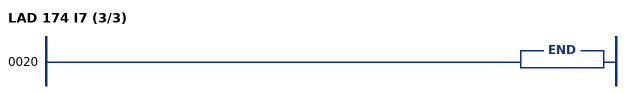
% Rung: 20 %
SOR END EOR

LADDER 175 "I7 RESULT"
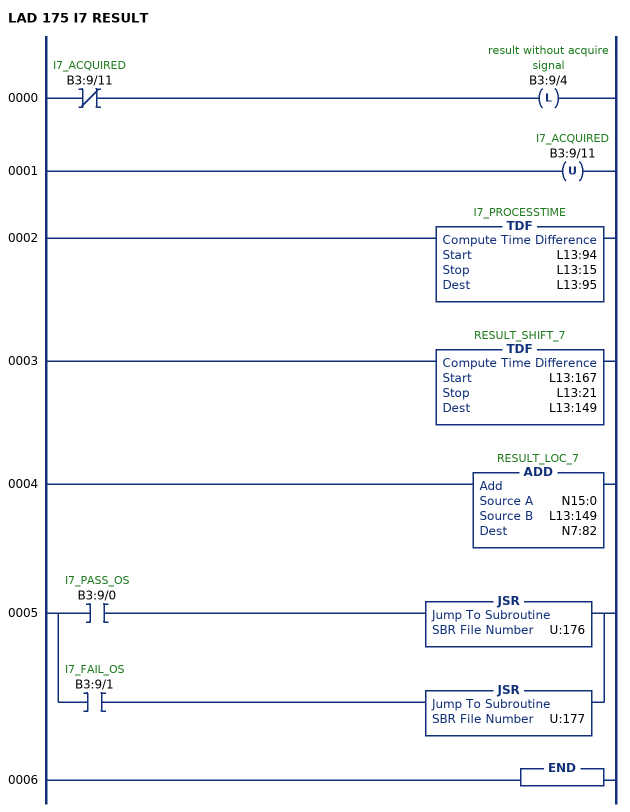
% Rung: 0 %
SOR XIO B3:9/11 OTL B3:9/4 EOR
%   B3:9/11  I7_ACQUIRED %
%   B3:9/4  "result without acquire signal" %
% Rung: 1 %
SOR OTU B3:9/11 EOR
%   B3:9/11  I7_ACQUIRED %
% Rung: 2 %
SOR TDF L13:94 L13:15 L13:95 EOR
%   L13:94  I7_TIMEOFACQ %
%   L13:15  THE_TIME %
%   L13:95  I7_PROCESSTIME %
% Rung: 3 %
SOR TDF L13:167 L13:21 L13:149 EOR
%   L13:167  I7_PROCESS_START_POS %
%   L13:21  TOP_POSITION %
%   L13:149  RESULT_SHIFT_7 %
% Rung: 4 %
SOR ADD N15:0 L13:149 N7:82 EOR
%   N15:0  I7_TRIG_LOC %
%   L13:149  RESULT_SHIFT_7 %
%   N7:82  RESULT_LOC_7 %
% Rung: 5 %
SOR BST XIC B3:9/0 JSR U:176 NXB XIC B3:9/1 JSR U:177 BND EOR
%   B3:9/0  I7_PASS_OS %
%   B3:9/1  I7_FAIL_OS %
% Rung: 6 %
SOR END EOR

LADDER 176 "I7 PASS"
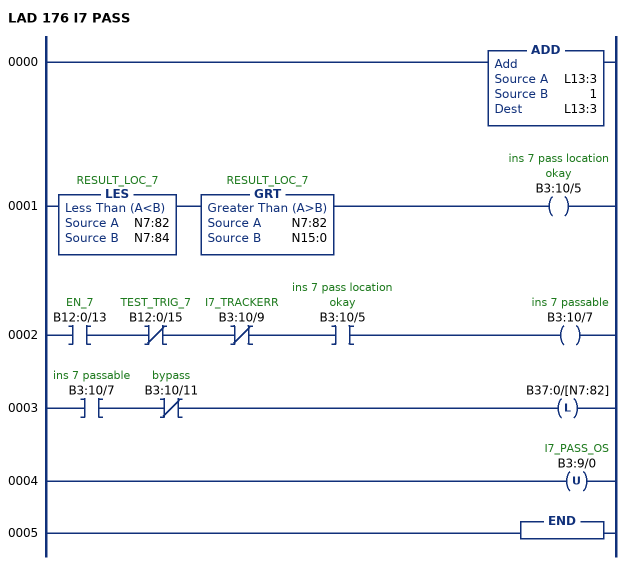
% Rung: 0 %
SOR ADD L13:3 1 L13:3 EOR
% Rung: 1 %
SOR LES N7:82 N7:84 GRT N7:82 N15:0 OTE B3:10/5 EOR
%   N7:82  RESULT_LOC_7 %
%   N7:84  I7_MAX_SHIFT %
%   N15:0  I7_TRIG_LOC %
%   B3:10/5  "ins 7 pass location okay" %
% Rung: 2 %
SOR XIC B12:0/13 XIO B12:0/15 XIO B3:10/9 XIC B3:10/5 OTE B3:10/7 EOR
%   B12:0/13  EN_7 %
%   B12:0/15  TEST_TRIG_7 %
%   B3:10/9  I7_TRACKERR %
%   B3:10/5  "ins 7 pass location okay" %
%   B3:10/7  "ins 7 passable" %
% Rung: 3 %
SOR XIC B3:10/7 XIO B3:10/11 OTL B37:0/[N7:82] EOR
%   B3:10/7  "ins 7 passable" %
%   B3:10/11  "bypass" %
%   B37:0  TOPGOOD1 %
%   N7:82  RESULT_LOC_7 %
% Rung: 4 %
SOR OTU B3:9/0 EOR
%   B3:9/0  I7_PASS_OS %
% Rung: 5 %
SOR END EOR

LADDER 177 "I7 FAIL"
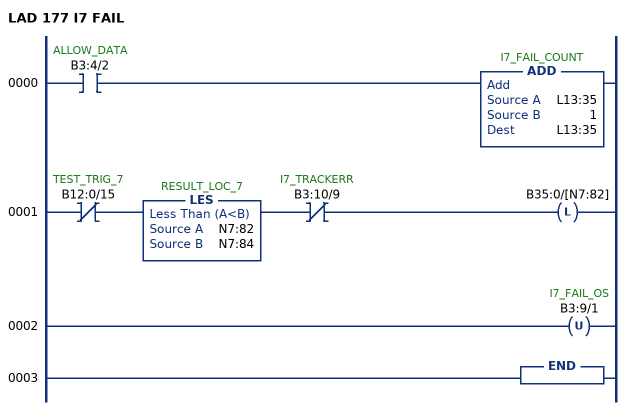
% Rung: 0 %
SOR XIC B3:4/2 ADD L13:35 1 L13:35 EOR
%   B3:4/2  ALLOW_DATA %
%   L13:35  I7_FAIL_COUNT %
% Rung: 1 %
SOR XIO B12:0/15 LES N7:82 N7:84 XIO B3:10/9 OTL B35:0/[N7:82] EOR
%   B12:0/15  TEST_TRIG_7 %
%   N7:82  RESULT_LOC_7 %
%   N7:84  I7_MAX_SHIFT %
%   B3:10/9  I7_TRACKERR %
%   B35:0  TOP_NG %
% Rung: 2 %
SOR OTU B3:9/1 EOR
%   B3:9/1  I7_FAIL_OS %
% Rung: 3 %
SOR END EOR

LADDER 178 "I7 ACQ"
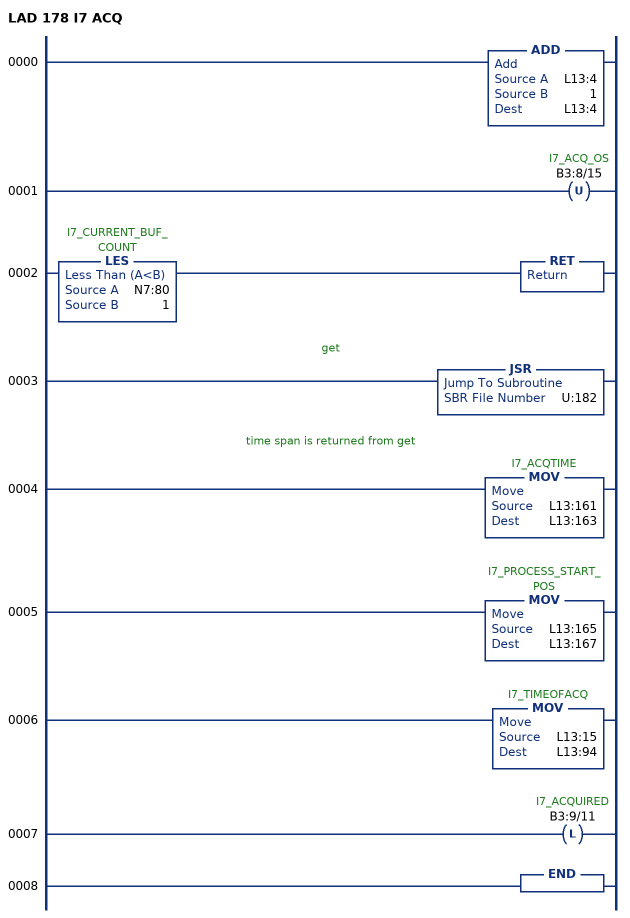
% Rung: 0 %
SOR ADD L13:4 1 L13:4 EOR
% Rung: 1 %
SOR OTU B3:8/15 EOR
%   B3:8/15  I7_ACQ_OS %
% Rung: 2 %
SOR LES N7:80 1 RET EOR
%   N7:80  I7_CURRENT_BUF_COUNT %
% Rung: 3 %
% get %
SOR JSR U:182 EOR
% Rung: 4 %
% time span is returned from get %
SOR MOV L13:161 L13:163 EOR
%   L13:161  I7_TIME_SPAN %
%   L13:163  I7_ACQTIME %
% Rung: 5 %
SOR MOV L13:165 L13:167 EOR
%   L13:165  I7_PULLED_POSITION %
%   L13:167  I7_PROCESS_START_POS %
% Rung: 6 %
SOR MOV L13:15 L13:94 EOR
%   L13:15  THE_TIME %
%   L13:94  I7_TIMEOFACQ %
% Rung: 7 %
SOR OTL B3:9/11 EOR
%   B3:9/11  I7_ACQUIRED %
% Rung: 8 %
SOR END EOR

LADDER 179 "I7 TESTER"
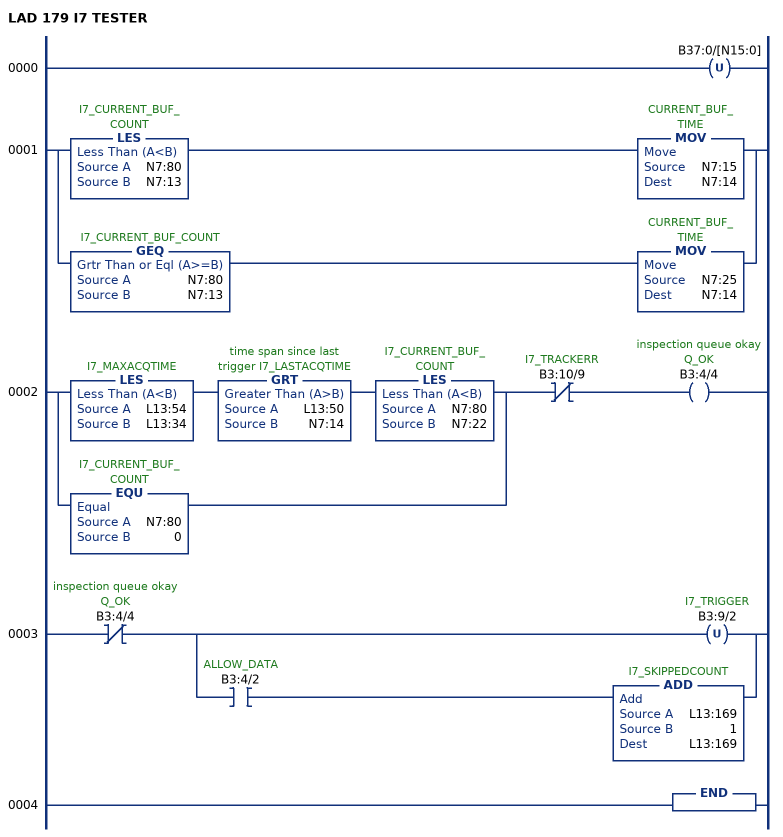
% Rung: 0 %
SOR OTU B37:0/[N15:0] EOR
%   B37:0  TOPGOOD1 %
%   N15:0  I7_TRIG_LOC %
% Rung: 1 %
SOR BST LES N7:80 N7:13 MOV N7:15 N7:14 NXB GEQ N7:80 N7:13 MOV N7:25 N7:14 BND EOR
%   N7:80  I7_CURRENT_BUF_COUNT %
%   N7:13  BUF_TRANS  "cam to pc buf transition" %
%   N7:15  CAM_BUF_TIME  "cam buf time" %
%   N7:14  CURRENT_BUF_TIME %
%   N7:25  PC_BUF_TIME  "pc buf time" %
% Rung: 2 %
SOR BST LES L13:54 L13:34 GRT L13:50 N7:14 LES N7:80 N7:22 NXB EQU N7:80 0 BND XIO B3:10/9 OTE B3:4/4 EOR
%   L13:54  I7_MAXACQTIME %
%   L13:34  MAX_ACQ_ALL  "absolute max acquire time before bypass trigger" %
%   L13:50  I7_LASTACQTIME  "time span since last trigger" %
%   N7:14  CURRENT_BUF_TIME %
%   N7:80  I7_CURRENT_BUF_COUNT %
%   N7:22  MAX_BUF_ALL  "max buffer count alowed before bypass" %
%   B3:10/9  I7_TRACKERR %
%   B3:4/4  Q_OK  "inspection queue okay" %
% Rung: 3 %
SOR XIO B3:4/4 BST OTU B3:9/2 NXB XIC B3:4/2 ADD L13:169 1 L13:169 BND EOR
%   B3:4/4  Q_OK  "inspection queue okay" %
%   B3:9/2  I7_TRIGGER %
%   B3:4/2  ALLOW_DATA %
%   L13:169  I7_SKIPPEDCOUNT %
% Rung: 4 %
SOR END EOR

LADDER 180 "I7 TRIG"
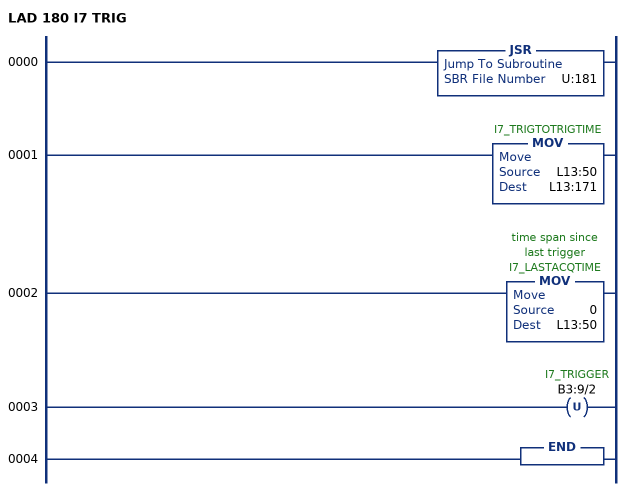
% Rung: 0 %
SOR JSR U:181 EOR
% Rung: 1 %
SOR MOV L13:50 L13:171 EOR
%   L13:50  I7_LASTACQTIME  "time span since last trigger" %
%   L13:171  I7_TRIGTOTRIGTIME %
% Rung: 2 %
SOR MOV 0 L13:50 EOR
%   L13:50  I7_LASTACQTIME  "time span since last trigger" %
% Rung: 3 %
SOR OTU B3:9/2 EOR
%   B3:9/2  I7_TRIGGER %
% Rung: 4 %
SOR END EOR

LADDER 181 "I7 FIFOSET"
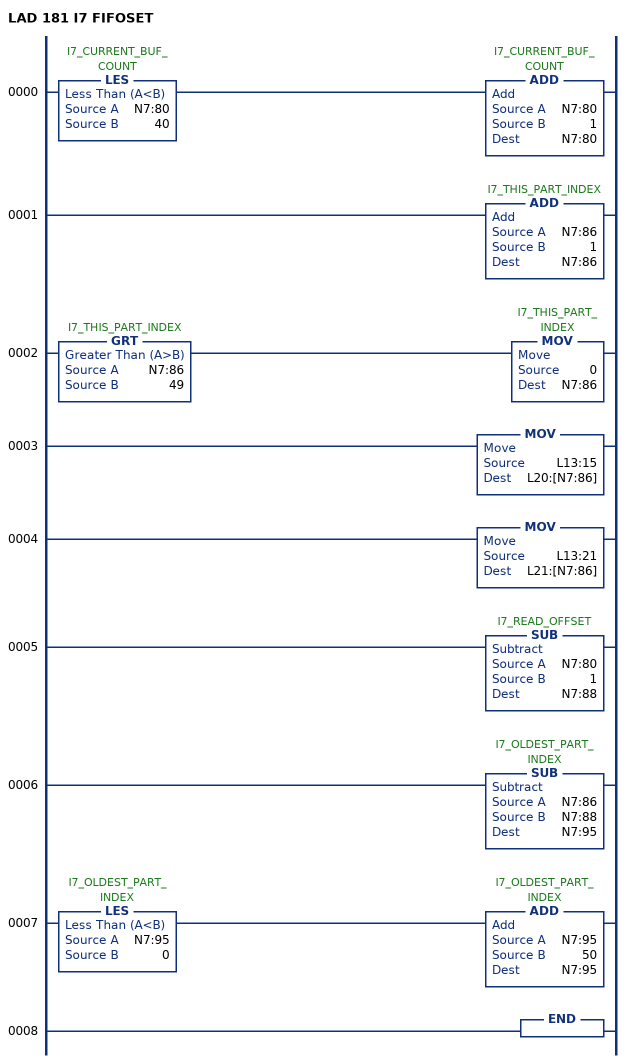
% Rung: 0 %
SOR LES N7:80 40 ADD N7:80 1 N7:80 EOR
%   N7:80  I7_CURRENT_BUF_COUNT %
% Rung: 1 %
SOR ADD N7:86 1 N7:86 EOR
%   N7:86  I7_THIS_PART_INDEX %
% Rung: 2 %
SOR GRT N7:86 49 MOV 0 N7:86 EOR
%   N7:86  I7_THIS_PART_INDEX %
% Rung: 3 %
SOR MOV L13:15 L20:[N7:86] EOR
%   L13:15  THE_TIME %
%   N7:86  I7_THIS_PART_INDEX %
% Rung: 4 %
SOR MOV L13:21 L21:[N7:86] EOR
%   L13:21  TOP_POSITION %
%   N7:86  I7_THIS_PART_INDEX %
% Rung: 5 %
SOR SUB N7:80 1 N7:88 EOR
%   N7:80  I7_CURRENT_BUF_COUNT %
%   N7:88  I7_READ_OFFSET %
% Rung: 6 %
SOR SUB N7:86 N7:88 N7:95 EOR
%   N7:86  I7_THIS_PART_INDEX %
%   N7:88  I7_READ_OFFSET %
%   N7:95  I7_OLDEST_PART_INDEX %
% Rung: 7 %
SOR LES N7:95 0 ADD N7:95 50 N7:95 EOR
%   N7:95  I7_OLDEST_PART_INDEX %
% Rung: 8 %
SOR END EOR

LADDER 182 "I7 FIFOGET"
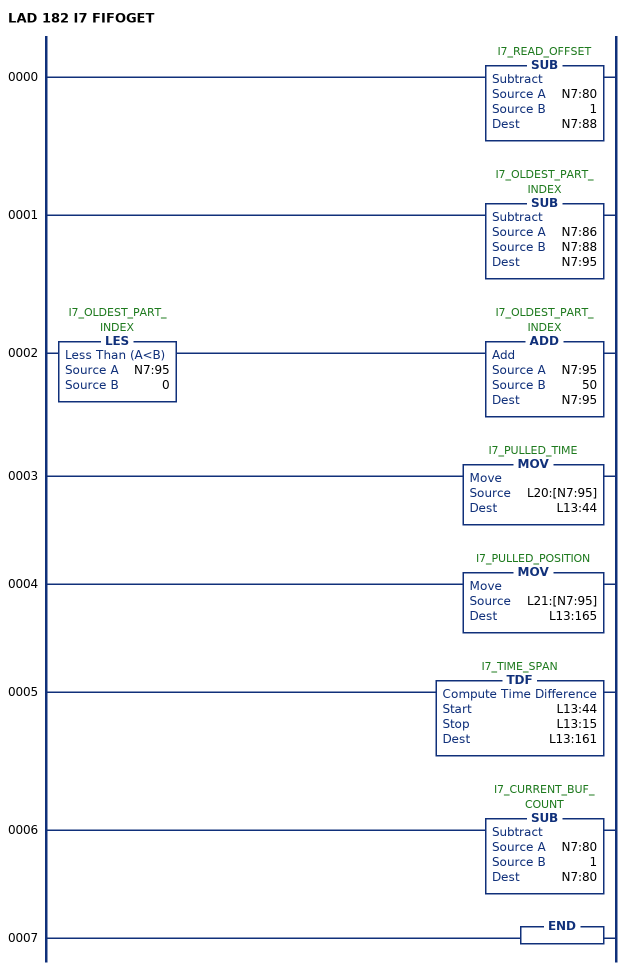
% Rung: 0 %
SOR SUB N7:80 1 N7:88 EOR
%   N7:80  I7_CURRENT_BUF_COUNT %
%   N7:88  I7_READ_OFFSET %
% Rung: 1 %
SOR SUB N7:86 N7:88 N7:95 EOR
%   N7:86  I7_THIS_PART_INDEX %
%   N7:88  I7_READ_OFFSET %
%   N7:95  I7_OLDEST_PART_INDEX %
% Rung: 2 %
SOR LES N7:95 0 ADD N7:95 50 N7:95 EOR
%   N7:95  I7_OLDEST_PART_INDEX %
% Rung: 3 %
SOR MOV L20:[N7:95] L13:44 EOR
%   N7:95  I7_OLDEST_PART_INDEX %
%   L13:44  I7_PULLED_TIME %
% Rung: 4 %
SOR MOV L21:[N7:95] L13:165 EOR
%   N7:95  I7_OLDEST_PART_INDEX %
%   L13:165  I7_PULLED_POSITION %
% Rung: 5 %
SOR TDF L13:44 L13:15 L13:161 EOR
%   L13:44  I7_PULLED_TIME %
%   L13:15  THE_TIME %
%   L13:161  I7_TIME_SPAN %
% Rung: 6 %
SOR SUB N7:80 1 N7:80 EOR
%   N7:80  I7_CURRENT_BUF_COUNT %
% Rung: 7 %
SOR END EOR

LADDER 183 "I7 DATA"
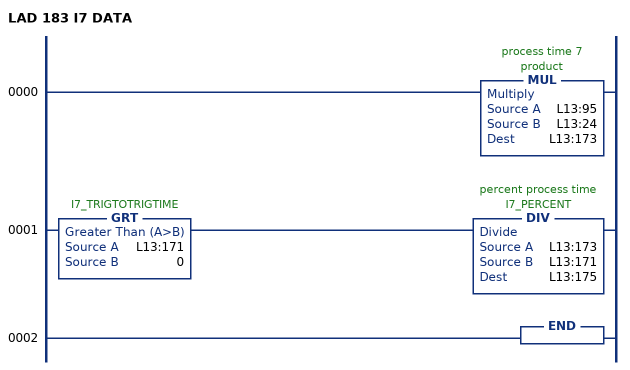
% Rung: 0 %
SOR MUL L13:95 L13:24 L13:173 EOR
%   L13:95  I7_PROCESSTIME %
%   L13:24  "multiplyer to make devision come out to a percentage" %
%   L13:173  "process time 7 product" %
% Rung: 1 %
SOR GRT L13:171 0 DIV L13:173 L13:171 L13:175 EOR
%   L13:171  I7_TRIGTOTRIGTIME %
%   L13:173  "process time 7 product" %
%   L13:175  I7_PERCENT  "percent process time" %
% Rung: 2 %
SOR END EOR

LADDER 184 "I7 FAULT"
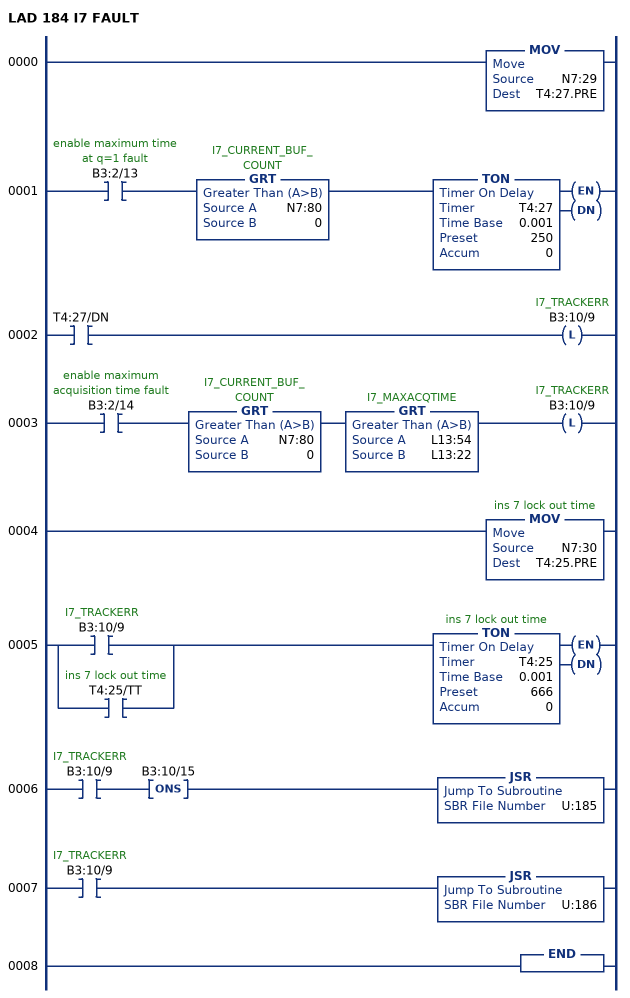
% Rung: 0 %
SOR MOV N7:29 T4:27.PRE EOR
%   N7:29  "max allowed ms time for q to be above 1 if safe fault is used" %
% Rung: 1 %
SOR XIC B3:2/13 GRT N7:80 0 TON T4:27 0.001 250 0 EOR
%   B3:2/13  "enable maximum time at q=1 fault" %
%   N7:80  I7_CURRENT_BUF_COUNT %
% Rung: 2 %
SOR XIC T4:27/DN OTL B3:10/9 EOR
%   B3:10/9  I7_TRACKERR %
% Rung: 3 %
SOR XIC B3:2/14 GRT N7:80 0 GRT L13:54 L13:22 OTL B3:10/9 EOR
%   B3:2/14  "enable maximum acquisition time fault" %
%   N7:80  I7_CURRENT_BUF_COUNT %
%   L13:54  I7_MAXACQTIME %
%   L13:22  "maximum of the longest acquire time allowed if maximum acquire time fault is enabled" %
%   B3:10/9  I7_TRACKERR %
% Rung: 4 %
SOR MOV N7:30 T4:25.PRE EOR
%   N7:30  "ms time setting to lock out inspection to give all pending images a chance to clear" %
%   T4:25  "ins 7 lock out time" %
% Rung: 5 %
SOR BST XIC B3:10/9 NXB XIC T4:25/TT BND TON T4:25 0.001 666 0 EOR
%   B3:10/9  I7_TRACKERR %
%   T4:25  "ins 7 lock out time" %
% Rung: 6 %
SOR XIC B3:10/9 ONS B3:10/15 JSR U:185 EOR
%   B3:10/9  I7_TRACKERR %
% Rung: 7 %
SOR XIC B3:10/9 JSR U:186 EOR
%   B3:10/9  I7_TRACKERR %
% Rung: 8 %
SOR END EOR

LADDER 185 "I7 FIX1"
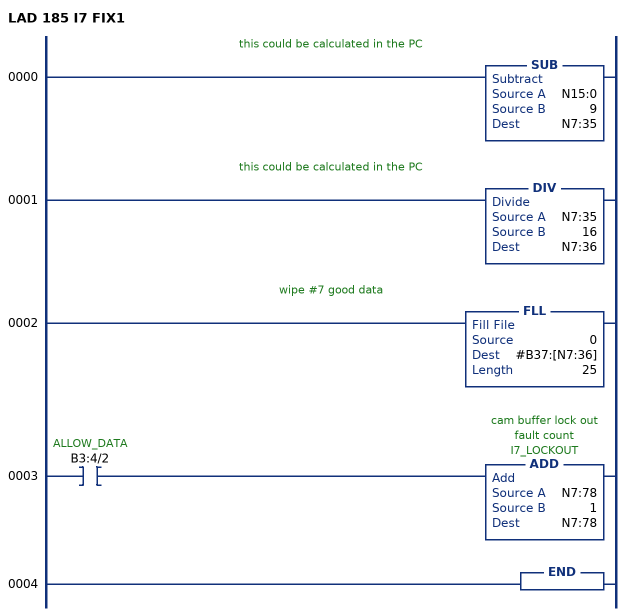
% Rung: 0 %
% this could be calculated in the PC %
SOR SUB N15:0 9 N7:35 EOR
%   N15:0  I7_TRIG_LOC %
% Rung: 1 %
% this could be calculated in the PC %
SOR DIV N7:35 16 N7:36 EOR
% Rung: 2 %
% wipe #7 good data %
SOR FLL 0 #B37:[N7:36] 25 EOR
% Rung: 3 %
SOR XIC B3:4/2 ADD N7:78 1 N7:78 EOR
%   B3:4/2  ALLOW_DATA %
%   N7:78  I7_LOCKOUT  "cam buffer lock out fault count" %
% Rung: 4 %
SOR END EOR

LADDER 186 "I7 FIX2"
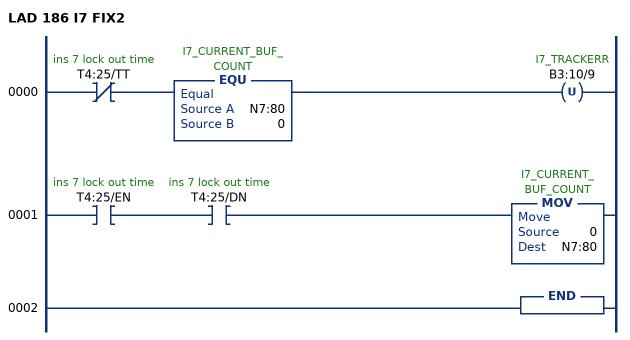
% Rung: 0 %
SOR XIO T4:25/TT EQU N7:80 0 OTU B3:10/9 EOR
%   T4:25  "ins 7 lock out time" %
%   N7:80  I7_CURRENT_BUF_COUNT %
%   B3:10/9  I7_TRACKERR %
% Rung: 1 %
SOR XIC T4:25/EN XIC T4:25/DN MOV 0 N7:80 EOR
%   T4:25  "ins 7 lock out time" %
%   N7:80  I7_CURRENT_BUF_COUNT %
% Rung: 2 %
SOR END EOR

LADDER 187 "I8"
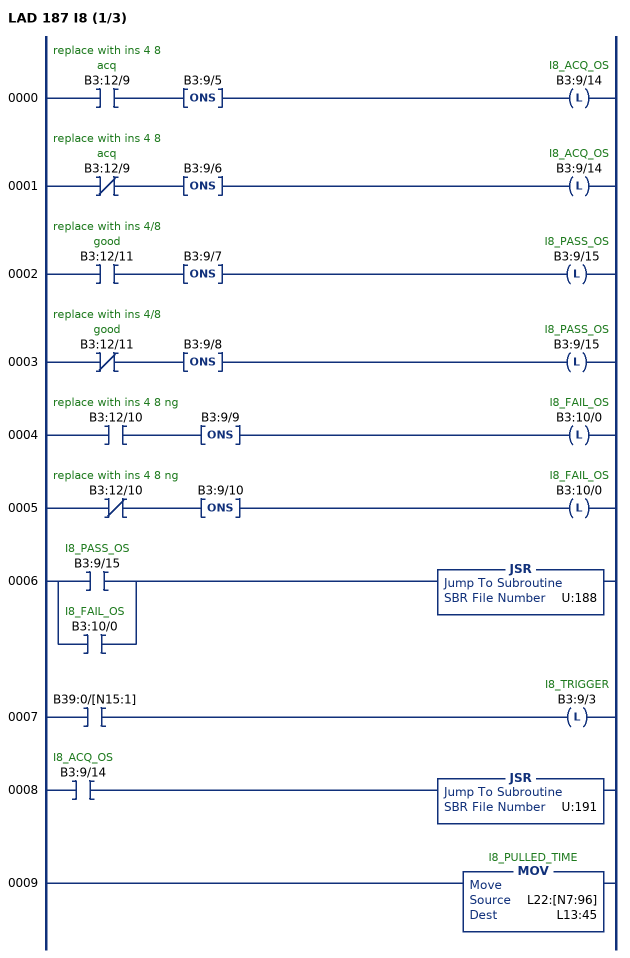
% Rung: 0 %
SOR XIC B3:12/9 ONS B3:9/5 OTL B3:9/14 EOR
%   B3:12/9  "replace with ins 4 8 acq" %
%   B3:9/14  I8_ACQ_OS %
% Rung: 1 %
SOR XIO B3:12/9 ONS B3:9/6 OTL B3:9/14 EOR
%   B3:12/9  "replace with ins 4 8 acq" %
%   B3:9/14  I8_ACQ_OS %
% Rung: 2 %
SOR XIC B3:12/11 ONS B3:9/7 OTL B3:9/15 EOR
%   B3:12/11  "replace with ins 4/8 good" %
%   B3:9/15  I8_PASS_OS %
% Rung: 3 %
SOR XIO B3:12/11 ONS B3:9/8 OTL B3:9/15 EOR
%   B3:12/11  "replace with ins 4/8 good" %
%   B3:9/15  I8_PASS_OS %
% Rung: 4 %
SOR XIC B3:12/10 ONS B3:9/9 OTL B3:10/0 EOR
%   B3:12/10  "replace with ins 4 8 ng" %
%   B3:10/0  I8_FAIL_OS %
% Rung: 5 %
SOR XIO B3:12/10 ONS B3:9/10 OTL B3:10/0 EOR
%   B3:12/10  "replace with ins 4 8 ng" %
%   B3:10/0  I8_FAIL_OS %
% Rung: 6 %
SOR BST XIC B3:9/15 NXB XIC B3:10/0 BND JSR U:188 EOR
%   B3:9/15  I8_PASS_OS %
%   B3:10/0  I8_FAIL_OS %
% Rung: 7 %
SOR XIC B39:0/[N15:1] OTL B3:9/3 EOR
%   B39:0  TOPGOOD2 %
%   N15:1  I8_TRIG_LOC %
%   B3:9/3  I8_TRIGGER %
% Rung: 8 %
SOR XIC B3:9/14 JSR U:191 EOR
%   B3:9/14  I8_ACQ_OS %
% Rung: 9 %
SOR MOV L22:[N7:96] L13:45 EOR
%   N7:96  I8_OLDEST_PART_INDEX %
%   L13:45  I8_PULLED_TIME %

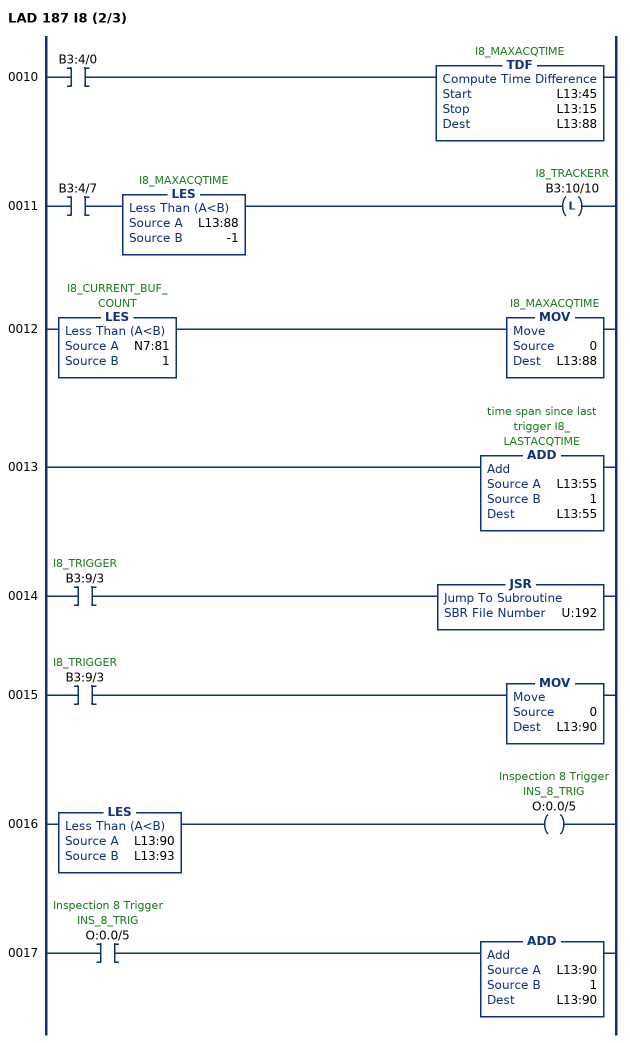
% Rung: 10 %
SOR XIC B3:4/0 TDF L13:45 L13:15 L13:88 EOR
%   L13:45  I8_PULLED_TIME %
%   L13:15  THE_TIME %
%   L13:88  I8_MAXACQTIME %
% Rung: 11 %
SOR XIC B3:4/7 LES L13:88 -1 OTL B3:10/10 EOR
%   L13:88  I8_MAXACQTIME %
%   B3:10/10  I8_TRACKERR %
% Rung: 12 %
SOR LES N7:81 1 MOV 0 L13:88 EOR
%   N7:81  I8_CURRENT_BUF_COUNT %
%   L13:88  I8_MAXACQTIME %
% Rung: 13 %
SOR ADD L13:55 1 L13:55 EOR
%   L13:55  I8_LASTACQTIME  "time span since last trigger" %
% Rung: 14 %
SOR XIC B3:9/3 JSR U:192 EOR
%   B3:9/3  I8_TRIGGER %
% Rung: 15 %
SOR XIC B3:9/3 MOV 0 L13:90 EOR
%   B3:9/3  I8_TRIGGER %
% Rung: 16 %
SOR LES L13:90 L13:93 OTE O:0.0/5 EOR
%   L13:93  "test fire count" %
%   O:0.0/5  INS_8_TRIG  "Inspection 8 Trigger" %
% Rung: 17 %
SOR XIC O:0.0/5 ADD L13:90 1 L13:90 EOR
%   O:0.0/5  INS_8_TRIG  "Inspection 8 Trigger" %

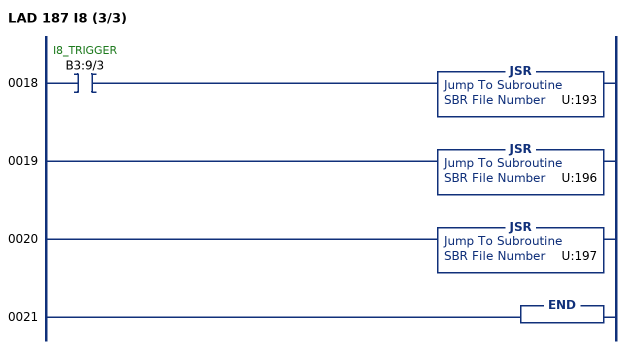
% Rung: 18 %
SOR XIC B3:9/3 JSR U:193 EOR
%   B3:9/3  I8_TRIGGER %
% Rung: 19 %
SOR JSR U:196 EOR
% Rung: 20 %
SOR JSR U:197 EOR
% Rung: 21 %
SOR END EOR

LADDER 188 "I8 RESULT"
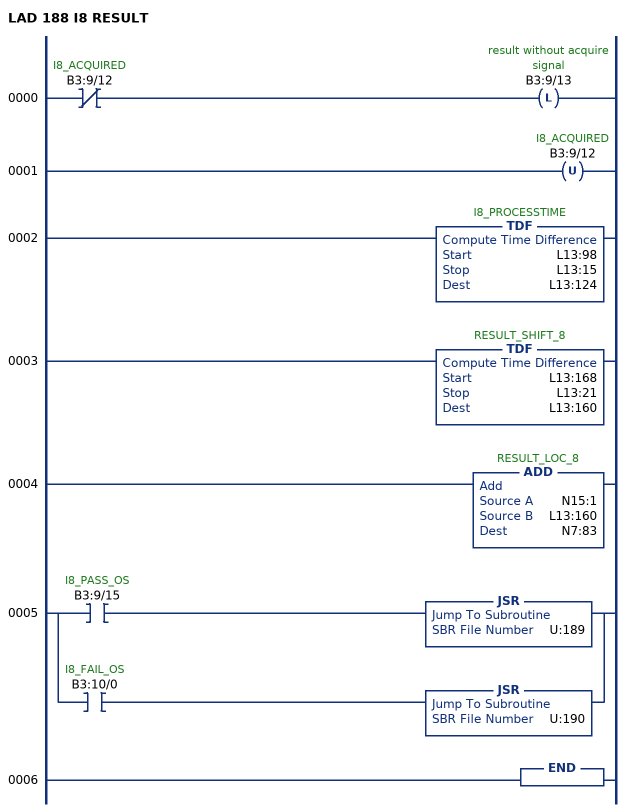
% Rung: 0 %
SOR XIO B3:9/12 OTL B3:9/13 EOR
%   B3:9/12  I8_ACQUIRED %
%   B3:9/13  "result without acquire signal" %
% Rung: 1 %
SOR OTU B3:9/12 EOR
%   B3:9/12  I8_ACQUIRED %
% Rung: 2 %
SOR TDF L13:98 L13:15 L13:124 EOR
%   L13:98  I8_TIMEOFACQ %
%   L13:15  THE_TIME %
%   L13:124  I8_PROCESSTIME %
% Rung: 3 %
SOR TDF L13:168 L13:21 L13:160 EOR
%   L13:168  I8_PROCESS_START_POS %
%   L13:21  TOP_POSITION %
%   L13:160  RESULT_SHIFT_8 %
% Rung: 4 %
SOR ADD N15:1 L13:160 N7:83 EOR
%   N15:1  I8_TRIG_LOC %
%   L13:160  RESULT_SHIFT_8 %
%   N7:83  RESULT_LOC_8 %
% Rung: 5 %
SOR BST XIC B3:9/15 JSR U:189 NXB XIC B3:10/0 JSR U:190 BND EOR
%   B3:9/15  I8_PASS_OS %
%   B3:10/0  I8_FAIL_OS %
% Rung: 6 %
SOR END EOR

LADDER 189 "I8 PASS"
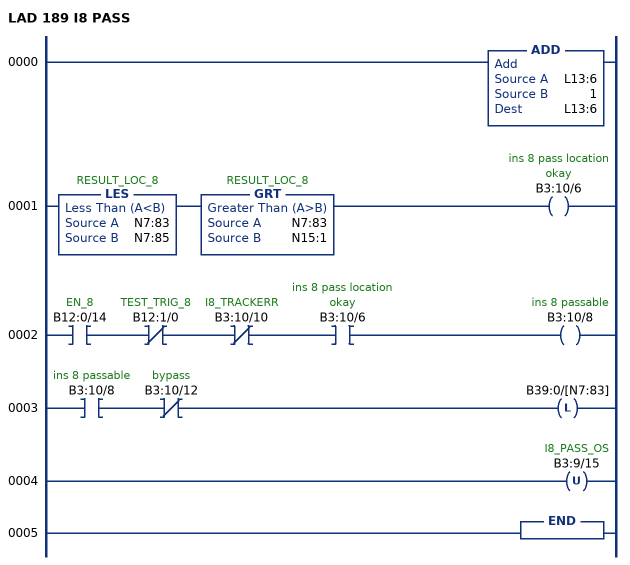
% Rung: 0 %
SOR ADD L13:6 1 L13:6 EOR
% Rung: 1 %
SOR LES N7:83 N7:85 GRT N7:83 N15:1 OTE B3:10/6 EOR
%   N7:83  RESULT_LOC_8 %
%   N7:85  I8_MAX_SHIFT %
%   N15:1  I8_TRIG_LOC %
%   B3:10/6  "ins 8 pass location okay" %
% Rung: 2 %
SOR XIC B12:0/14 XIO B12:1/0 XIO B3:10/10 XIC B3:10/6 OTE B3:10/8 EOR
%   B12:0/14  EN_8 %
%   B12:1/0  TEST_TRIG_8 %
%   B3:10/10  I8_TRACKERR %
%   B3:10/6  "ins 8 pass location okay" %
%   B3:10/8  "ins 8 passable" %
% Rung: 3 %
SOR XIC B3:10/8 XIO B3:10/12 OTL B39:0/[N7:83] EOR
%   B3:10/8  "ins 8 passable" %
%   B3:10/12  "bypass" %
%   B39:0  TOPGOOD2 %
%   N7:83  RESULT_LOC_8 %
% Rung: 4 %
SOR OTU B3:9/15 EOR
%   B3:9/15  I8_PASS_OS %
% Rung: 5 %
SOR END EOR

LADDER 190 "I8 FAIL"
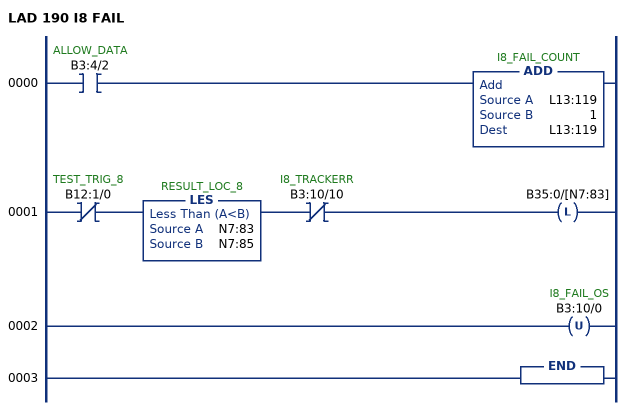
% Rung: 0 %
SOR XIC B3:4/2 ADD L13:119 1 L13:119 EOR
%   B3:4/2  ALLOW_DATA %
%   L13:119  I8_FAIL_COUNT %
% Rung: 1 %
SOR XIO B12:1/0 LES N7:83 N7:85 XIO B3:10/10 OTL B35:0/[N7:83] EOR
%   B12:1/0  TEST_TRIG_8 %
%   N7:83  RESULT_LOC_8 %
%   N7:85  I8_MAX_SHIFT %
%   B3:10/10  I8_TRACKERR %
%   B35:0  TOP_NG %
% Rung: 2 %
SOR OTU B3:10/0 EOR
%   B3:10/0  I8_FAIL_OS %
% Rung: 3 %
SOR END EOR

LADDER 191 "I8 ACQ"
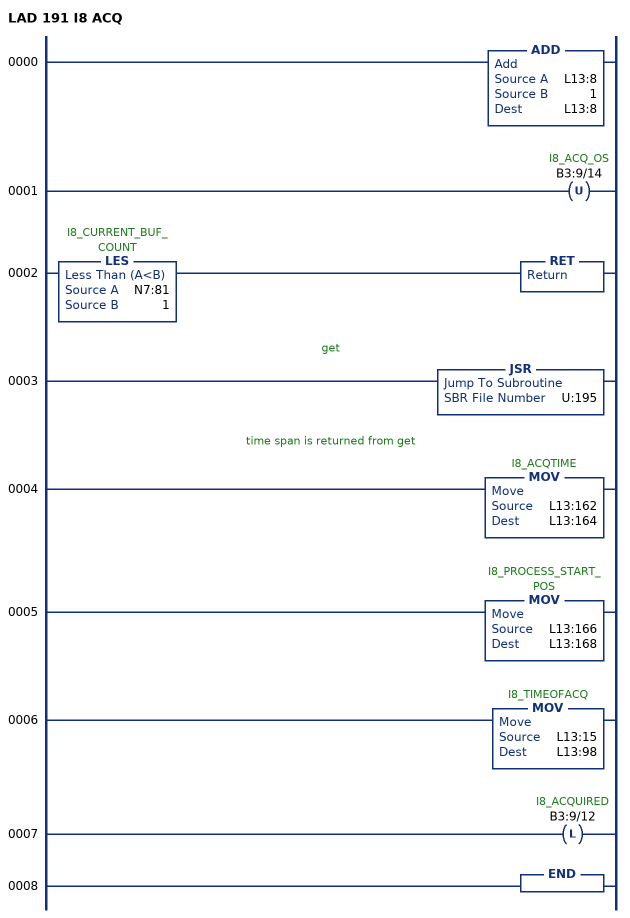
% Rung: 0 %
SOR ADD L13:8 1 L13:8 EOR
% Rung: 1 %
SOR OTU B3:9/14 EOR
%   B3:9/14  I8_ACQ_OS %
% Rung: 2 %
SOR LES N7:81 1 RET EOR
%   N7:81  I8_CURRENT_BUF_COUNT %
% Rung: 3 %
% get %
SOR JSR U:195 EOR
% Rung: 4 %
% time span is returned from get %
SOR MOV L13:162 L13:164 EOR
%   L13:162  I8_TIME_SPAN %
%   L13:164  I8_ACQTIME %
% Rung: 5 %
SOR MOV L13:166 L13:168 EOR
%   L13:166  I8_PULLED_POSITION %
%   L13:168  I8_PROCESS_START_POS %
% Rung: 6 %
SOR MOV L13:15 L13:98 EOR
%   L13:15  THE_TIME %
%   L13:98  I8_TIMEOFACQ %
% Rung: 7 %
SOR OTL B3:9/12 EOR
%   B3:9/12  I8_ACQUIRED %
% Rung: 8 %
SOR END EOR

LADDER 192 "I8 TESTER"
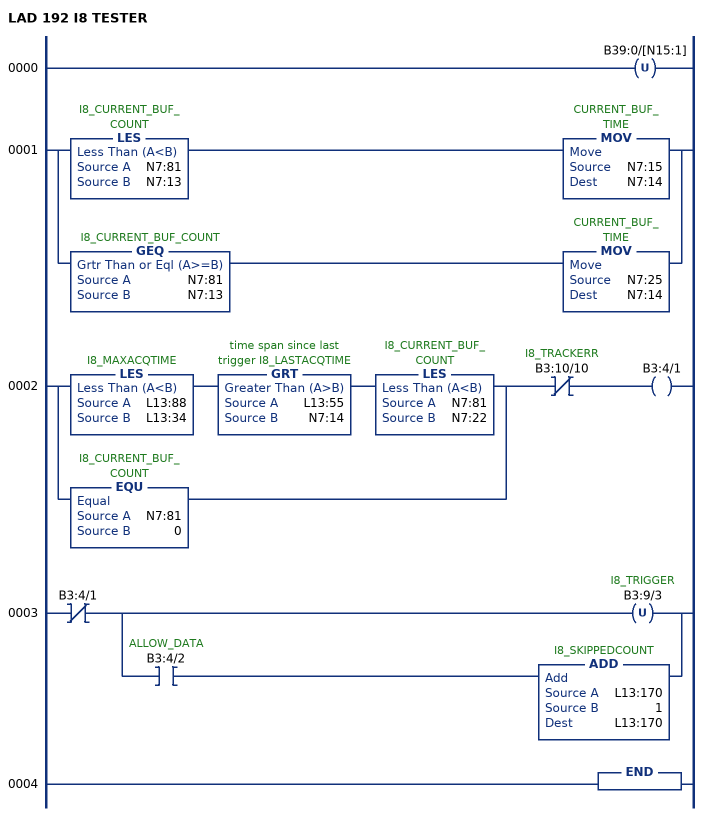
% Rung: 0 %
SOR OTU B39:0/[N15:1] EOR
%   B39:0  TOPGOOD2 %
%   N15:1  I8_TRIG_LOC %
% Rung: 1 %
SOR BST LES N7:81 N7:13 MOV N7:15 N7:14 NXB GEQ N7:81 N7:13 MOV N7:25 N7:14 BND EOR
%   N7:81  I8_CURRENT_BUF_COUNT %
%   N7:13  BUF_TRANS  "cam to pc buf transition" %
%   N7:15  CAM_BUF_TIME  "cam buf time" %
%   N7:14  CURRENT_BUF_TIME %
%   N7:25  PC_BUF_TIME  "pc buf time" %
% Rung: 2 %
SOR BST LES L13:88 L13:34 GRT L13:55 N7:14 LES N7:81 N7:22 NXB EQU N7:81 0 BND XIO B3:10/10 OTE B3:4/1 EOR
%   L13:88  I8_MAXACQTIME %
%   L13:34  MAX_ACQ_ALL  "absolute max acquire time before bypass trigger" %
%   L13:55  I8_LASTACQTIME  "time span since last trigger" %
%   N7:14  CURRENT_BUF_TIME %
%   N7:81  I8_CURRENT_BUF_COUNT %
%   N7:22  MAX_BUF_ALL  "max buffer count alowed before bypass" %
%   B3:10/10  I8_TRACKERR %
% Rung: 3 %
SOR XIO B3:4/1 BST OTU B3:9/3 NXB XIC B3:4/2 ADD L13:170 1 L13:170 BND EOR
%   B3:9/3  I8_TRIGGER %
%   B3:4/2  ALLOW_DATA %
%   L13:170  I8_SKIPPEDCOUNT %
% Rung: 4 %
SOR END EOR

LADDER 193 "I8 TRIG"
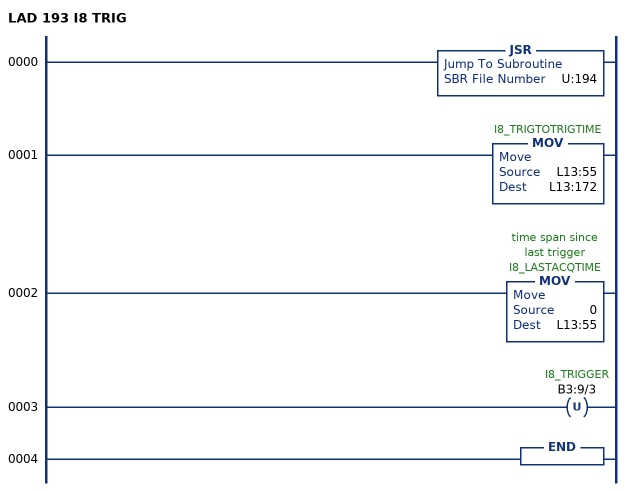
% Rung: 0 %
SOR JSR U:194 EOR
% Rung: 1 %
SOR MOV L13:55 L13:172 EOR
%   L13:55  I8_LASTACQTIME  "time span since last trigger" %
%   L13:172  I8_TRIGTOTRIGTIME %
% Rung: 2 %
SOR MOV 0 L13:55 EOR
%   L13:55  I8_LASTACQTIME  "time span since last trigger" %
% Rung: 3 %
SOR OTU B3:9/3 EOR
%   B3:9/3  I8_TRIGGER %
% Rung: 4 %
SOR END EOR

LADDER 194 "I8 FIFOSET"
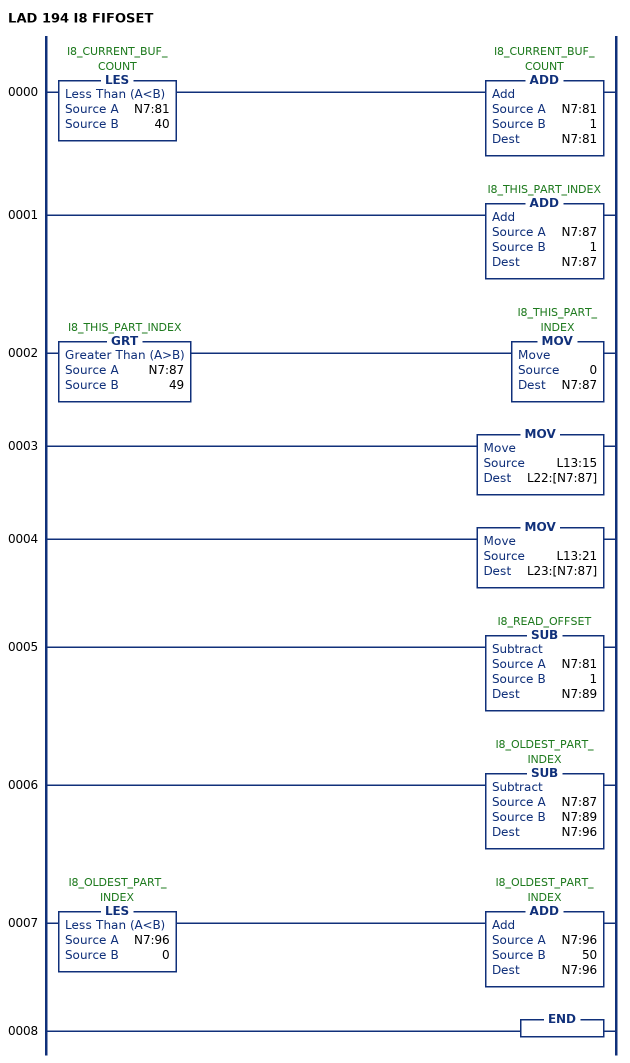
% Rung: 0 %
SOR LES N7:81 40 ADD N7:81 1 N7:81 EOR
%   N7:81  I8_CURRENT_BUF_COUNT %
% Rung: 1 %
SOR ADD N7:87 1 N7:87 EOR
%   N7:87  I8_THIS_PART_INDEX %
% Rung: 2 %
SOR GRT N7:87 49 MOV 0 N7:87 EOR
%   N7:87  I8_THIS_PART_INDEX %
% Rung: 3 %
SOR MOV L13:15 L22:[N7:87] EOR
%   L13:15  THE_TIME %
%   N7:87  I8_THIS_PART_INDEX %
% Rung: 4 %
SOR MOV L13:21 L23:[N7:87] EOR
%   L13:21  TOP_POSITION %
%   N7:87  I8_THIS_PART_INDEX %
% Rung: 5 %
SOR SUB N7:81 1 N7:89 EOR
%   N7:81  I8_CURRENT_BUF_COUNT %
%   N7:89  I8_READ_OFFSET %
% Rung: 6 %
SOR SUB N7:87 N7:89 N7:96 EOR
%   N7:87  I8_THIS_PART_INDEX %
%   N7:89  I8_READ_OFFSET %
%   N7:96  I8_OLDEST_PART_INDEX %
% Rung: 7 %
SOR LES N7:96 0 ADD N7:96 50 N7:96 EOR
%   N7:96  I8_OLDEST_PART_INDEX %
% Rung: 8 %
SOR END EOR

LADDER 195 "I8 FIFOGET"
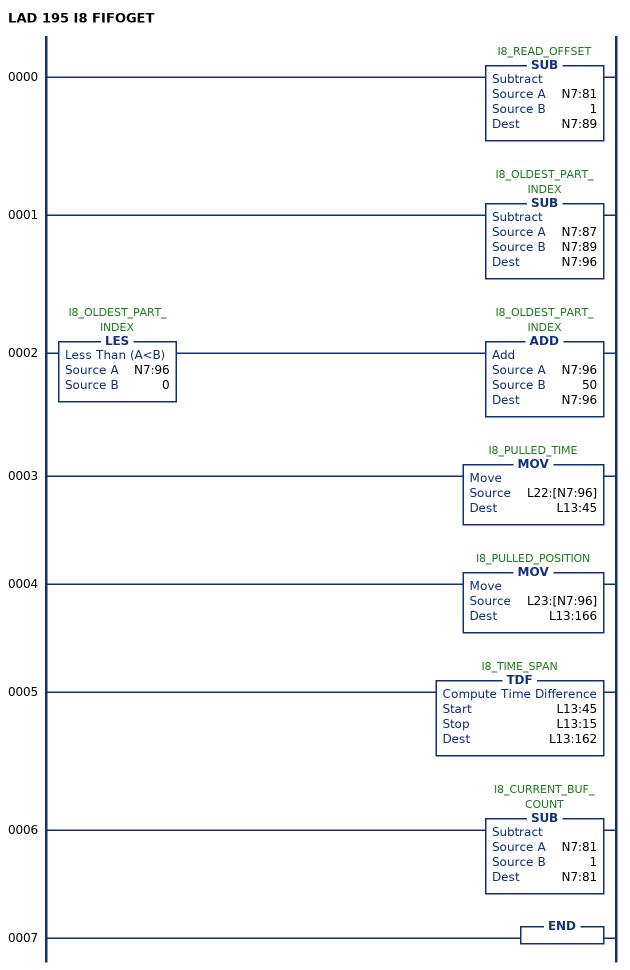
% Rung: 0 %
SOR SUB N7:81 1 N7:89 EOR
%   N7:81  I8_CURRENT_BUF_COUNT %
%   N7:89  I8_READ_OFFSET %
% Rung: 1 %
SOR SUB N7:87 N7:89 N7:96 EOR
%   N7:87  I8_THIS_PART_INDEX %
%   N7:89  I8_READ_OFFSET %
%   N7:96  I8_OLDEST_PART_INDEX %
% Rung: 2 %
SOR LES N7:96 0 ADD N7:96 50 N7:96 EOR
%   N7:96  I8_OLDEST_PART_INDEX %
% Rung: 3 %
SOR MOV L22:[N7:96] L13:45 EOR
%   N7:96  I8_OLDEST_PART_INDEX %
%   L13:45  I8_PULLED_TIME %
% Rung: 4 %
SOR MOV L23:[N7:96] L13:166 EOR
%   N7:96  I8_OLDEST_PART_INDEX %
%   L13:166  I8_PULLED_POSITION %
% Rung: 5 %
SOR TDF L13:45 L13:15 L13:162 EOR
%   L13:45  I8_PULLED_TIME %
%   L13:15  THE_TIME %
%   L13:162  I8_TIME_SPAN %
% Rung: 6 %
SOR SUB N7:81 1 N7:81 EOR
%   N7:81  I8_CURRENT_BUF_COUNT %
% Rung: 7 %
SOR END EOR

LADDER 196 "I8 DATA"
